// TIA Portal V20 export
TYPE "typeAxisPositionCondition"
// stored: Access Published, Namespace LER
   STRUCT
      interlockOk : Array[0..15] of Bool;
      interlockError : Array[0..15] of Bool;
      intOut : Array[0..9] of Bool;
   END_STRUCT;
END_TYPE
